// TwinCAT 3 PLC project PLC
// ProgramVersion: 3.1.4026.15
// libraries:
//   Tc2_Standard, * (Beckhoff Automation GmbH)
//   Tc2_System, * (Beckhoff Automation GmbH)
// project tree:
//   / PlcTask.TcTTO
//   POUs/ MAIN.TcPOU
// real-time tasks:
//   TASK PlcTask: cycle T#10ms, priority 20, ADS port 350

CONFIGURATION PLC
    RESOURCE PLC ON TwinCAT3
        TASK PlcTask(INTERVAL := T#10ms, PRIORITY := 20);
        PROGRAM MAIN WITH PlcTask : MAIN;
    END_RESOURCE
END_CONFIGURATION

// ---- POUs/MAIN.TcPOU
PROGRAM MAIN
VAR
	bStartCmd		: BOOL;
	bStopCmd		: BOOL;
	fSpeedCmd		: LREAL;
	bRunning		: BOOL;
	fSpeedAct		: LREAL;
	sName			: STRING := 'My React Faceplate';
END_VAR

IF bStartCmd AND NOT bRunning THEN
	bRunning := TRUE;
END_IF

IF bStopCmd AND bRunning THEN
	bRunning := FALSE;
END_IF

IF bRunning THEN 
	IF fSpeedAct < fSpeedCmd THEN
		fSpeedAct := fSpeedAct + 0.25;
	END_IF
	IF fSpeedAct > fSpeedCmd THEN
		fSpeedAct := fSpeedAct - 0.25;
	END_IF
END_IF

IF NOT bRunning THEN
	IF fSpeedAct > 0 THEN
		fSpeedAct := fSpeedAct - 0.25;
	END_IF
	IF fSpeedAct < 0 THEN
		fSpeedAct := 0;
	END_IF
END_IF

END_PROGRAM
